// TIA Portal V20 export
FUNCTION "EM4_TeachingData" : Void   // FC83, LAD
// stored: Namespace Unit1.Em4, SetENOAutomatically false
BEGIN

REGION Network 2 (SCL): SideTape FixStage AxisX Teaching Position
   // SideTape FixStage AxisX Position 0
   "Unit1.Em4.HmiInterface".cmSideTapeFixStageAxisX.configuration.setPositions[0].position := 330.0;
   "Unit1.Em4.HmiInterface".cmSideTapeFixStageAxisX.configuration.setPositions[0].velocity := 10.0;

   // SideTape FixStage AxisX Position 1
   "Unit1.Em4.HmiInterface".cmSideTapeFixStageAxisX.configuration.setPositions[1].position := 16.46;
   "Unit1.Em4.HmiInterface".cmSideTapeFixStageAxisX.configuration.setPositions[1].velocity := 10.0;

   // SideTape FixStage AxisX Position 2
   "Unit1.Em4.HmiInterface".cmSideTapeFixStageAxisX.configuration.setPositions[2].position := 330.0;
   "Unit1.Em4.HmiInterface".cmSideTapeFixStageAxisX.configuration.setPositions[2].velocity := 10.0;


   /////////// ZONE //////////

   // SideTape FixStage AxisX Position 9
   "Unit1.Em4.HmiInterface".cmSideTapeFixStageAxisX.configuration.setPositions[9].position := 16.46;
   "Unit1.Em4.HmiInterface".cmSideTapeFixStageAxisX.configuration.setPositions[9].velocity := 10.0;
END_REGION

REGION Network 3 (SCL): SideTape FixStage AxisC Teaching Position
   // SideTape FixStage AxisC Position 0
   "Unit1.Em4.HmiInterface".cmSideTapeFixStageAxisC.configuration.setPositions[0].position := 90.0;
   "Unit1.Em4.HmiInterface".cmSideTapeFixStageAxisC.configuration.setPositions[0].velocity := 10.0;

   // SideTape FixStage AxisC Position 1
   "Unit1.Em4.HmiInterface".cmSideTapeFixStageAxisC.configuration.setPositions[1].position := 180.0;
   "Unit1.Em4.HmiInterface".cmSideTapeFixStageAxisC.configuration.setPositions[1].velocity := 10.0;

   // SideTape FixStage AxisC Position 2
   "Unit1.Em4.HmiInterface".cmSideTapeFixStageAxisC.configuration.setPositions[2].position := 0.0;
   "Unit1.Em4.HmiInterface".cmSideTapeFixStageAxisC.configuration.setPositions[2].velocity := 10.0;

   // SideTape FixStage AxisC Position 3
   "Unit1.Em4.HmiInterface".cmSideTapeFixStageAxisC.configuration.setPositions[3].position := -90.0;
   "Unit1.Em4.HmiInterface".cmSideTapeFixStageAxisC.configuration.setPositions[3].velocity := 10.0;
END_REGION

REGION Network 4 (SCL): SideTape Attachment AxisX Teaching Position
   //SideTape Attachment AxisX Position 0
   "Unit1.Em4.HmiInterface".cmSideTapeAttachmentAxisX.configuration.setPositions[0].position := 469.0;
   "Unit1.Em4.HmiInterface".cmSideTapeAttachmentAxisX.configuration.setPositions[0].velocity := 10.0;
   "Unit1.Em4.HmiInterface".cmSideTapeAttachmentAxisX.configuration.setPositions[0].acceleration := 100.0;
   "Unit1.Em4.HmiInterface".cmSideTapeAttachmentAxisX.configuration.setPositions[0].deceleration := 100.0;

   //SideTape Attachment AxisX Position 1
   "Unit1.Em4.HmiInterface".cmSideTapeAttachmentAxisX.configuration.setPositions[1].position := 469.0;
   "Unit1.Em4.HmiInterface".cmSideTapeAttachmentAxisX.configuration.setPositions[1].velocity := 10.0;
   "Unit1.Em4.HmiInterface".cmSideTapeAttachmentAxisX.configuration.setPositions[1].acceleration := 100.0;
   "Unit1.Em4.HmiInterface".cmSideTapeAttachmentAxisX.configuration.setPositions[1].deceleration := 100.0;

   //SideTape Attachment AxisX Position 2
   "Unit1.Em4.HmiInterface".cmSideTapeAttachmentAxisX.configuration.setPositions[2].position := 610.0;
   "Unit1.Em4.HmiInterface".cmSideTapeAttachmentAxisX.configuration.setPositions[2].velocity := 10.0;
   "Unit1.Em4.HmiInterface".cmSideTapeAttachmentAxisX.configuration.setPositions[2].acceleration := 100.0;
   "Unit1.Em4.HmiInterface".cmSideTapeAttachmentAxisX.configuration.setPositions[2].deceleration := 100.0;

   //SideTape Attachment AxisX Position 3
   "Unit1.Em4.HmiInterface".cmSideTapeAttachmentAxisX.configuration.setPositions[3].position := 116.0;
   "Unit1.Em4.HmiInterface".cmSideTapeAttachmentAxisX.configuration.setPositions[3].velocity := 10.0;
   "Unit1.Em4.HmiInterface".cmSideTapeAttachmentAxisX.configuration.setPositions[3].acceleration := 100.0;
   "Unit1.Em4.HmiInterface".cmSideTapeAttachmentAxisX.configuration.setPositions[3].deceleration := 100.0;

   //SideTape Attachment AxisX Position 4
   "Unit1.Em4.HmiInterface".cmSideTapeAttachmentAxisX.configuration.setPositions[4].position := 37.0;
   "Unit1.Em4.HmiInterface".cmSideTapeAttachmentAxisX.configuration.setPositions[4].velocity := 10.0;



   //SideTape Attachment AxisX Position 5
   "Unit1.Em4.HmiInterface".cmSideTapeAttachmentAxisX.configuration.setPositions[5].position := 42.4;
   "Unit1.Em4.HmiInterface".cmSideTapeAttachmentAxisX.configuration.setPositions[5].velocity := 10.0;



   //SideTape Attachment AxisX Position 6
   "Unit1.Em4.HmiInterface".cmSideTapeAttachmentAxisX.configuration.setPositions[6].position := 40.5;
   "Unit1.Em4.HmiInterface".cmSideTapeAttachmentAxisX.configuration.setPositions[6].velocity := 10.0;


   ////////////////////// ZONE //////////////////////

   //SideTape Attachment AxisX Position 7
   "Unit1.Em4.HmiInterface".cmSideTapeAttachmentAxisX.configuration.setPositions[7].position := 400.0;
   "Unit1.Em4.HmiInterface".cmSideTapeAttachmentAxisX.configuration.setPositions[7].velocity := 10.0;



   //SideTape Attachment AxisX Position 8
   "Unit1.Em4.HmiInterface".cmSideTapeAttachmentAxisX.configuration.setPositions[8].position := 450.0;
   "Unit1.Em4.HmiInterface".cmSideTapeAttachmentAxisX.configuration.setPositions[8].velocity := 10.0;



   //SideTape Attachment AxisX Position 9
   "Unit1.Em4.HmiInterface".cmSideTapeAttachmentAxisX.configuration.setPositions[9].position := 40.4;
   "Unit1.Em4.HmiInterface".cmSideTapeAttachmentAxisX.configuration.setPositions[9].velocity := 10.0;
END_REGION

REGION Network 5 (SCL): SideTape Attachment AxisY Teaching Position
   //SideTape Attachment AxisY Position 0
   "Unit1.Em4.HmiInterface".cmSideTapeAttachmentAxisY.configuration.setPositions[0].position := 0.0;
   "Unit1.Em4.HmiInterface".cmSideTapeAttachmentAxisY.configuration.setPositions[0].velocity := 10.0;

   //SideTape Attachment AxisY Position 1
   "Unit1.Em4.HmiInterface".cmSideTapeAttachmentAxisY.configuration.setPositions[1].position := 100.0;
   "Unit1.Em4.HmiInterface".cmSideTapeAttachmentAxisY.configuration.setPositions[1].velocity := 10.0;
   "Unit1.Em4.HmiInterface".cmSideTapeAttachmentAxisY.configuration.setPositions[1].acceleration := 100.0;
   "Unit1.Em4.HmiInterface".cmSideTapeAttachmentAxisY.configuration.setPositions[1].deceleration := 100.0;

   //SideTape Attachment AxisY Position 2
   "Unit1.Em4.HmiInterface".cmSideTapeAttachmentAxisY.configuration.setPositions[2].position := 110.0;
   "Unit1.Em4.HmiInterface".cmSideTapeAttachmentAxisY.configuration.setPositions[2].velocity := 10.0;


   //SideTape Attachment AxisY Position 3
   "Unit1.Em4.HmiInterface".cmSideTapeAttachmentAxisY.configuration.setPositions[3].position := 210.0;
   "Unit1.Em4.HmiInterface".cmSideTapeAttachmentAxisY.configuration.setPositions[3].velocity := 10.0;



   //SideTape Attachment AxisY Position 4
   "Unit1.Em4.HmiInterface".cmSideTapeAttachmentAxisY.configuration.setPositions[4].position := 220.0;
   "Unit1.Em4.HmiInterface".cmSideTapeAttachmentAxisY.configuration.setPositions[4].velocity := 10.0;

   //SideTape Attachment AxisY Position 5
   "Unit1.Em4.HmiInterface".cmSideTapeAttachmentAxisY.configuration.setPositions[5].position := 230.0;
   "Unit1.Em4.HmiInterface".cmSideTapeAttachmentAxisY.configuration.setPositions[5].velocity := 10.0;

   //SideTape Attachment AxisY Position 6
   "Unit1.Em4.HmiInterface".cmSideTapeAttachmentAxisY.configuration.setPositions[6].position := 240.0;
   "Unit1.Em4.HmiInterface".cmSideTapeAttachmentAxisY.configuration.setPositions[6].velocity := 10.0;


   ////////////////////// ZONE //////////////////////

   //SideTape Attachment AxisY Position 7
   "Unit1.Em4.HmiInterface".cmSideTapeAttachmentAxisY.configuration.setPositions[7].position := 50.0;
   "Unit1.Em4.HmiInterface".cmSideTapeAttachmentAxisY.configuration.setPositions[7].velocity := 10.0;

   //SideTape Attachment AxisY Position 8
   "Unit1.Em4.HmiInterface".cmSideTapeAttachmentAxisY.configuration.setPositions[8].position := 60.0;
   "Unit1.Em4.HmiInterface".cmSideTapeAttachmentAxisY.configuration.setPositions[8].velocity := 10.0;

   //SideTape Attachment AxisY Position 9
   "Unit1.Em4.HmiInterface".cmSideTapeAttachmentAxisY.configuration.setPositions[9].position := 0.0;
   "Unit1.Em4.HmiInterface".cmSideTapeAttachmentAxisY.configuration.setPositions[9].velocity := 10.0;
END_REGION
END_FUNCTION
